TYPE ST_SafetyOut :
STRUCT
    stMCCStatusOut: ST_MCCStatusOut;
    stMCC_CustomStatusOut: ST_MCC_CustomStatusOut;
    astSafetyFunctionOut: ARRAY[1..GVL_SafetyIO.cNBR_OF_SF] OF ST_SafetyFunctionOut;

    bSTOActive: BOOL;
    bTechnosoftMotionErrors: BOOL;
END_STRUCT
END_TYPE

(* stored: Version 1.1.0.1
   DUT ST_SafetyOut: Id {d70660d3-487b-0b0c-33db-774882ada2f1} *)
